// TIA Portal project "Sorting_Basic" (V19)
// Vorlageprojekt für das Buch mit Zielsystem S7-1200

(* hardware
DEVICE "S7-1200-Station_1"  S7-1200 Station
   slot 0: "Baugruppenträger_0"  Rack  V1.0
   slot 1: "PLC_1"  CPU 1211C DC/DC/DC  6ES7 211-1AE40-0XB0  V4.1
*)

// ===== PLC "PLC_1"  CPU 1211C DC/DC/DC =====

VAR_GLOBAL   // PLC tag table "Standard-Variablentabelle"
   "Load" AT %Q0.1 : Bool;
   "Running" AT %M0.0 : Bool;
   "Loaded_Marker" AT %M0.1 : Bool;
   "Mem+Pallet" AT %M0.2 : Bool;
   "Mem-Pallet" AT %M0.3 : Bool;
   "Loading_Stage" AT %M0.4 : Bool;
   "Tag_2" AT %M0.5 : Bool;
   "Tag_3" AT %M0.6 : Bool;
   "Load Conv Start" AT %M0.7 : Bool;
   "CD_Counter" AT %M1.0 : Bool;
   "Left_path" AT %M1.1 : Bool;
   "Right_path" AT %M1.2 : Bool;
   "At_Left_Entry+" AT %M1.3 : Bool;
   "Tag_7" AT %M1.7 : Bool;
   "Pallet +" AT %M1.4 : Bool;
   "At_Left_Exit-" AT %M1.5 : Bool;
   "Stop_Conv_Left" AT %M1.6 : Bool;
   "At_Left_Entry-" AT %M2.0 : Bool;
   "Start_Left_Conv" AT %M2.1 : Bool;
   "Tag_1" AT %M2.2 : Bool;
   "Stop_Transfer_Right" AT %M2.3 : Bool;
   "Tag_4" AT %M2.4 : Bool;
   "Start_Right_Conv" AT %M2.5 : Bool;
   "Tag_6" AT %M2.6 : Bool;
   "Stop_Conv_Right" AT %M2.7 : Bool;
   "CD right entry" AT %M3.0 : Bool;
   "CD left entry" AT %M3.1 : Bool;
   "CD_Counter(1)" AT %M3.2 : Bool;
   "Tag_8" AT %M3.3 : Bool;
   "Tag_5" AT %M4.0 : Bool;
   "Tag_9" AT %M4.7 : Bool;
END_VAR

VAR_GLOBAL   // PLC tag table "Tag table from XML_1"
   "High sensor" AT %I0.0 : Bool;
   "Low sensor" AT %I0.1 : Bool;
   "Pallet sensor" AT %I0.2 : Bool;
   "Loaded" AT %I0.3 : Bool;
   "At left entry" AT %I0.4 : Bool;
   "At left exit" AT %I0.5 : Bool;
   "At right entry" AT %I0.6 : Bool;
   "At right exit" AT %I0.7 : Bool;
   "Start" AT %I1.0 : Bool;
   "Reset" AT %I1.1 : Bool;
   "Stop" AT %I1.2 : Bool;
   "Emergency stop" AT %I1.3 : Bool;
   "Auto" AT %I1.4 : Bool;
   "FACTORY I/O (Running)" AT %I1.5 : Bool;
   "Conveyor entry" AT %Q0.0 : Bool;
   "Unload" AT %Q0.2 : Bool;
   "Transf. left" AT %Q0.3 : Bool;
   "Transf. right" AT %Q0.4 : Bool;
   "Conveyor left" AT %Q0.5 : Bool;
   "Conveyor right" AT %Q0.6 : Bool;
   "Start light" AT %Q0.7 : Bool;
   "Reset light" AT %Q1.0 : Bool;
   "Stop light" AT %Q1.1 : Bool;
   "Counter" AT %QW30 : Int;
END_VAR

// folder: System blocks/Program resources

DATA_BLOCK "IEC_Counter_0_DB_2"   // DB3
{ S7_Optimized_Access := 'TRUE' }
AUTHOR : Simatic
FAMILY : IEC
NAME : CNTR
VERSION : 1.0
// stored: InstanceOfName IEC_COUNTER
"IEC_COUNTER"
BEGIN
END_DATA_BLOCK

// folder: (top level)

FUNCTION "MHJ-PLC-Lab-Function-S71200" : Void   // FC9000, SCL
{ S7_Optimized_Access := 'TRUE' }
VERSION : 0.1
   VAR_TEMP
      rdTimeReturn : Int;
      outputTime : DTL;
      SyncVal : Byte;
      forVal : Int;
      forVal_2 : Int;
      Value : Byte;
   END_VAR
   VAR CONSTANT
      CompVal : Byte := 16#34;
      Value_01 : Byte := 16#11;
      Value_01_DW : DWord := 16#A165_D992;
      Value_02_DW : DWord := 16#58BE_4401;
   END_VAR
BEGIN

   #Value:=PEEK(area := 16#82,
        dbNumber := 0,
        byteOffset := 511);
   #Value := #Value + 1;

   POKE(area := 16#82,
        dbNumber := 0,
        byteOffset := 511,
        value := #Value);

   POKE(area:=16#81,
        dbNumber:=0,
        byteOffset:=1016,
        value:=#Value_01_DW);
   POKE(area := 16#81,
        dbNumber := 0,
        byteOffset := 1020,
        value := #Value_02_DW);

   POKE(area := 16#81,
        dbNumber := 0,
        byteOffset := 511,
        value := B#16#00);

   FOR #forVal := 0 TO 120 DO
       FOR #forVal_2:=0 TO 10 DO
           #rdTimeReturn:=RD_SYS_T(#outputTime);
           #rdTimeReturn := WR_SYS_T(#outputTime);
           #rdTimeReturn := RD_SYS_T(#outputTime);
           #rdTimeReturn := WR_SYS_T(#outputTime);
       END_FOR;
       #SyncVal:= PEEK(area := 16#81,
                      dbNumber := 0,
                      byteOffset := 511);
       IF #SyncVal = #CompVal THEN
          GOTO M_1;
       END_IF;
   END_FOR;
   RETURN;

   M_1:
   POKE(area := 16#81,
        dbNumber := 0,
        byteOffset := 511,
        value := B#16#0);
END_FUNCTION

ORGANIZATION_BLOCK "Main"   // OB1, LAD, ProgramCycle
TITLE = "Main Program Sweep (Cycle)"
{ S7_Optimized_Access := 'TRUE' }
VERSION : 0.1
   VAR_INPUT
      Initial_Call : Bool;   // Initial call of this OB
      Remanence : Bool;   // =True, if remanent data are available
   END_VAR
   VAR_TEMP   // added for the SCL form of the ladder/FBD networks
      _w1 : Bool;
      _w2 : Bool;
      _w3 : Bool;
   END_VAR
BEGIN

REGION Network 1: Konnektierungsbaustein für PLC-Lab
   // Im Netzwerk 1 wird der Konnektierungsbaustein für PLC-Lab aufgerufen.
   // Dieser Aufruf darf nicht entfernt werden!
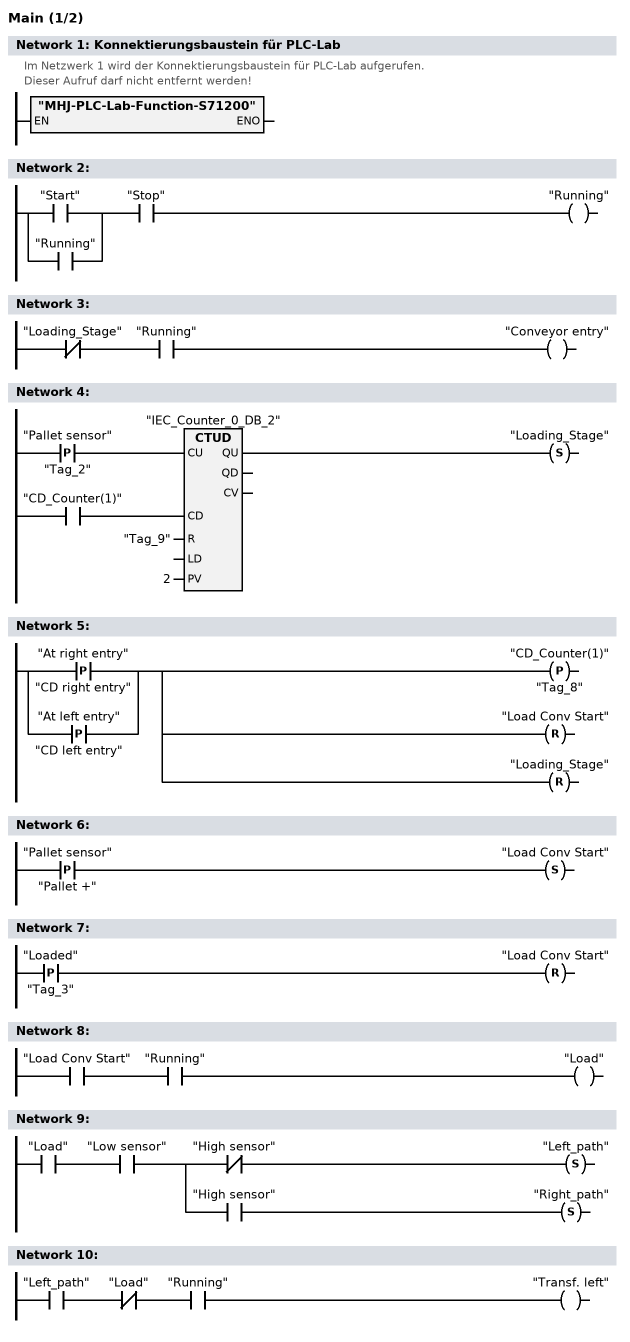
   RUNG wire#powerrail
      "MHJ-PLC-Lab-Function-S71200"()
   END_RUNG
   // the same network as SCL:
   "MHJ-PLC-Lab-Function-S71200"();
END_REGION

REGION Network 2
   RUNG wire#powerrail
      Contact( "Start" )
      wire#w1
      Contact( "Stop" )
      Coil( "Running" )
   END_RUNG
   RUNG wire#powerrail
      Contact( "Running" )
   END_RUNG wire#w1
   // the same network as SCL:
   "Running" := ("Start" OR "Running") AND "Stop";
END_REGION

REGION Network 3
   RUNG wire#powerrail
      I_Contact( "Loading_Stage" )
      Contact( "Running" )
      Coil( "Conveyor entry" )
   END_RUNG
   // the same network as SCL:
   "Conveyor entry" := NOT "Loading_Stage" AND "Running";
END_REGION

REGION Network 4
   #_w1 := "Pallet sensor" AND NOT "Tag_2";   // rising edge of "Pallet sensor"
   "Tag_2" := "Pallet sensor";
   "IEC_Counter_0_DB_2".CTUD(CU := #_w1, CD := "CD_Counter(1)", R := "Tag_9", PV := 2);
   IF "IEC_Counter_0_DB_2".QU THEN "Loading_Stage" := TRUE; END_IF;
END_REGION

REGION Network 5
   #_w1 := "At right entry" AND NOT "CD right entry";   // rising edge of "At right entry"
   "CD right entry" := "At right entry";
   #_w2 := "At left entry" AND NOT "CD left entry";   // rising edge of "At left entry"
   "CD left entry" := "At left entry";
   #_w3 := #_w1 OR #_w2;
   "CD_Counter(1)" := #_w3 AND NOT "Tag_8";   // rising edge
   "Tag_8" := #_w3;
   IF #_w3 THEN
       "Load Conv Start" := FALSE;
       "Loading_Stage" := FALSE;
   END_IF;
END_REGION

REGION Network 6
   RUNG wire#powerrail
      P_Contact(operand := "Pallet sensor", bit := "Pallet +")
      S_Coil( "Load Conv Start" )
   END_RUNG
   // the same network as SCL:
   #_w1 := "Pallet sensor" AND NOT "Pallet +";   // rising edge of "Pallet sensor"
   "Pallet +" := "Pallet sensor";
   IF #_w1 THEN "Load Conv Start" := TRUE; END_IF;
END_REGION

REGION Network 7
   RUNG wire#powerrail
      P_Contact(operand := "Loaded", bit := "Tag_3")
      R_Coil( "Load Conv Start" )
   END_RUNG
   // the same network as SCL:
   #_w1 := "Loaded" AND NOT "Tag_3";   // rising edge of "Loaded"
   "Tag_3" := "Loaded";
   IF #_w1 THEN "Load Conv Start" := FALSE; END_IF;
END_REGION

REGION Network 8
   RUNG wire#powerrail
      Contact( "Load Conv Start" )
      Contact( "Running" )
      Coil( "Load" )
   END_RUNG
   // the same network as SCL:
   "Load" := "Load Conv Start" AND "Running";
END_REGION

REGION Network 9
   RUNG wire#powerrail
      Contact( "Load" )
      Contact( "Low sensor" )
      wire#w1
      I_Contact( "High sensor" )
      S_Coil( "Left_path" )
   END_RUNG
   RUNG wire#w1
      Contact( "High sensor" )
      S_Coil( "Right_path" )
   END_RUNG
   // the same network as SCL:
   #_w1 := "Load" AND "Low sensor";
   IF #_w1 AND NOT "High sensor" THEN "Left_path" := TRUE; END_IF;
   IF #_w1 AND "High sensor" THEN "Right_path" := TRUE; END_IF;
END_REGION

REGION Network 10
   RUNG wire#powerrail
      Contact( "Left_path" )
      I_Contact( "Load" )
      Contact( "Running" )
      Coil( "Transf. left" )
   END_RUNG
   // the same network as SCL:
   "Transf. left" := "Left_path" AND NOT "Load" AND "Running";
END_REGION

REGION Network 11
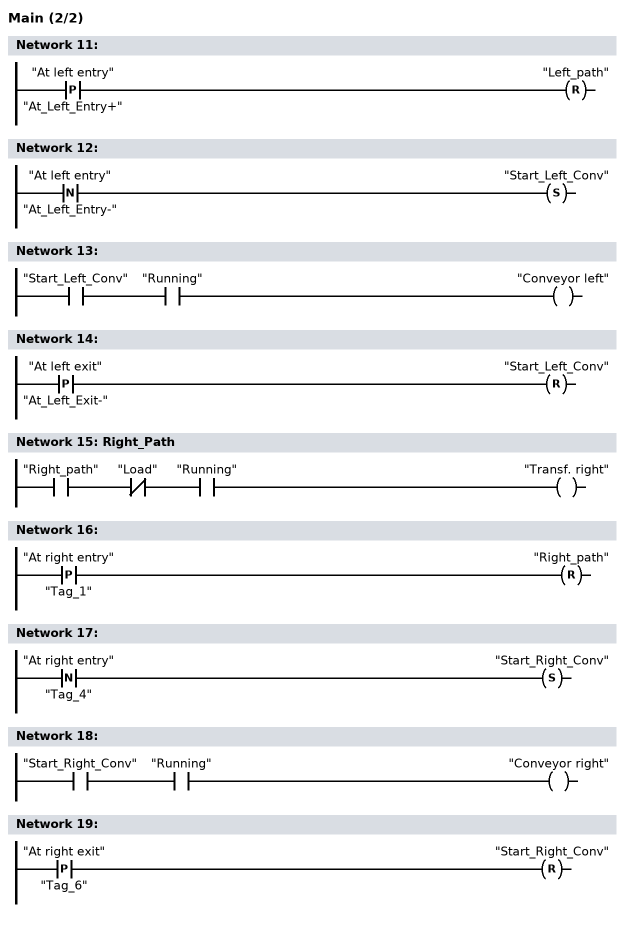
   RUNG wire#powerrail
      P_Contact(operand := "At left entry", bit := "At_Left_Entry+")
      R_Coil( "Left_path" )
   END_RUNG
   // the same network as SCL:
   #_w1 := "At left entry" AND NOT "At_Left_Entry+";   // rising edge of "At left entry"
   "At_Left_Entry+" := "At left entry";
   IF #_w1 THEN "Left_path" := FALSE; END_IF;
END_REGION

REGION Network 12
   RUNG wire#powerrail
      N_Contact(operand := "At left entry", bit := "At_Left_Entry-")
      S_Coil( "Start_Left_Conv" )
   END_RUNG
   // the same network as SCL:
   #_w1 := NOT "At left entry" AND "At_Left_Entry-";   // falling edge of "At left entry"
   "At_Left_Entry-" := "At left entry";
   IF #_w1 THEN "Start_Left_Conv" := TRUE; END_IF;
END_REGION

REGION Network 13
   RUNG wire#powerrail
      Contact( "Start_Left_Conv" )
      Contact( "Running" )
      Coil( "Conveyor left" )
   END_RUNG
   // the same network as SCL:
   "Conveyor left" := "Start_Left_Conv" AND "Running";
END_REGION

REGION Network 14
   RUNG wire#powerrail
      P_Contact(operand := "At left exit", bit := "At_Left_Exit-")
      R_Coil( "Start_Left_Conv" )
   END_RUNG
   // the same network as SCL:
   #_w1 := "At left exit" AND NOT "At_Left_Exit-";   // rising edge of "At left exit"
   "At_Left_Exit-" := "At left exit";
   IF #_w1 THEN "Start_Left_Conv" := FALSE; END_IF;
END_REGION

REGION Network 15: Right_Path
   RUNG wire#powerrail
      Contact( "Right_path" )
      I_Contact( "Load" )
      Contact( "Running" )
      Coil( "Transf. right" )
   END_RUNG
   // the same network as SCL:
   "Transf. right" := "Right_path" AND NOT "Load" AND "Running";
END_REGION

REGION Network 16
   RUNG wire#powerrail
      P_Contact(operand := "At right entry", bit := "Tag_1")
      R_Coil( "Right_path" )
   END_RUNG
   // the same network as SCL:
   #_w1 := "At right entry" AND NOT "Tag_1";   // rising edge of "At right entry"
   "Tag_1" := "At right entry";
   IF #_w1 THEN "Right_path" := FALSE; END_IF;
END_REGION

REGION Network 17
   RUNG wire#powerrail
      N_Contact(operand := "At right entry", bit := "Tag_4")
      S_Coil( "Start_Right_Conv" )
   END_RUNG
   // the same network as SCL:
   #_w1 := NOT "At right entry" AND "Tag_4";   // falling edge of "At right entry"
   "Tag_4" := "At right entry";
   IF #_w1 THEN "Start_Right_Conv" := TRUE; END_IF;
END_REGION

REGION Network 18
   RUNG wire#powerrail
      Contact( "Start_Right_Conv" )
      Contact( "Running" )
      Coil( "Conveyor right" )
   END_RUNG
   // the same network as SCL:
   "Conveyor right" := "Start_Right_Conv" AND "Running";
END_REGION

REGION Network 19
   RUNG wire#powerrail
      P_Contact(operand := "At right exit", bit := "Tag_6")
      R_Coil( "Start_Right_Conv" )
   END_RUNG
   // the same network as SCL:
   #_w1 := "At right exit" AND NOT "Tag_6";   // rising edge of "At right exit"
   "Tag_6" := "At right exit";
   IF #_w1 THEN "Start_Right_Conv" := FALSE; END_IF;
END_REGION
END_ORGANIZATION_BLOCK